Omron Sysmac Studio project AA_Festo (Sysmac Studio 1.60.0.64010, StandardProject)

# Controller Right_PLC: NX1P2-9B24DT1 version 1.42
Task PrimaryTask (priority 4, period or condition 4000): Main, Comunication_FINS
Library OEN_Communication_V1_0_22 1.0.22 (contents left out)
Library FINS_NX 1.1.0 (contents left out)

VAR_GLOBAL
    trama : ARRAY[0..3] OF OEN\Modbus\sModbusReq := [(Enable := True, NodeAdr := 1, FunctionCode := Fn15_WriteMultipleCoils, Read := (StartAddressRemote := 0, StartAddressLocal := 0, Count := 0), Write := (StartAddressRemote := 0, StartAddressLocal := 0, Count := 40)), (Enable := True, NodeAdr := 1, FunctionCode := Fn02_ReadDiscreteInputs, Read := (StartAddressRemote := 0, StartAddressLocal := 0, Count := 40), Write := (StartAddressRemote := 0, StartAddressLocal := 0, Count := 0)), (Enable := True, NodeAdr := 1, FunctionCode := Fn04_ReadInputRegisters, Read := (StartAddressRemote := 0, StartAddressLocal := 0, Count := 5), Write := (StartAddressRemote := 0, StartAddressLocal := 0, Count := 0)), (Enable := True, NodeAdr := 1, FunctionCode := Fn16_WriteMultipleRegisters, Read := (StartAddressRemote := 0, StartAddressLocal := 0, Count := 0), Write := (StartAddressRemote := 0, StartAddressLocal := 0, Count := 5))];
    out_Dig : ARRAY[0..99] OF BOOL;  (* Out_Digitais; [0] Emitter base; [1] Pneumatico inicio; [3] Motor Tapete; [4] Positioner Clamp; [5] Positioner raise (Stop Peça); [19] start button light A1; [8] Positioner Clamp extra; [9] Avanço Pneumatico Vácuo; [10] Baixa Pneumatico Vácuo; [11] Vácuo; [21] reset button light A1; [14] garra prende; [7] Emitter top; [15] Plataforma Frente; [16] Plataforma Tras; [20] stop button light A1; [17] Remover; [23] Start Button Light A2; [24] Stop Button Light A2; [25] Reset Button Light A2; [33] Reset Factory *)
    in_Dig : ARRAY[0..99] OF BOOL;  (* Entradas_Digitais; [1] Sensor Pneumático Trás; [0] Sensor Deteta Peça Base; [2] Sensor Pneumático Frente; [4] Sensor Inicio Tapete; [5] Sensor Leitura Cor; [8] Sensor Fim Tapete; [13] Sensor Vácuo Pneumatico cima; [10] Sensor Positioner clamp extra; [11] Sensor Vácuo Pneumatico  Frente; [6] Sensor Positioner raise; [23] Sensor Plataforma Trás; [17] Sensor Posição Recolha; [19] Sensor Posição Despeço Esquerda; [21] Sensor Garra Prende; [20] Sensor Posição Despejo Direita; [22] Sensor Plataforma Frente; [26] Stop Button A1; [25] Start Button A1; [14] Sensor Vácuo; [7] Sensor Positioner clamp; [12] Sensor Vácuo Pneumatico Trás; [18] Sensor Barra Início; [27] Reset Button A1; [29] Start Button A2; [30] Stop Button A2; [31] Reset Button A2; [33] Sensor Garra Cima; [34] Sensor Garra Baixo *)
    in_Analog : ARRAY[0..20] OF WORD;  (* Entradas_Analogicas *)
    out_analog : ARRAY[0..20] OF WORD;  (* Saidas_analogicas; [1] Garra y; [0] Garra x; [2] Garra Z *)
    A2_Start : BOOL;  (* at BuiltInIO://cpu/#0/Input_Bit_08 *)
    A2_Stop : BOOL;  (* at BuiltInIO://cpu/#0/Input_Bit_09 *)
    A2_Reset : BOOL;  (* at BuiltInIO://cpu/#0/Input_Bit_11 *)
    A2_Chave : BOOL;  (* at BuiltInIO://cpu/#0/Input_Bit_10 *)
    A2_S_PR : BOOL;  (* Sensor Posição Recolha; at BuiltInIO://cpu/#0/Input_Bit_00 *)
    A2_S_GC : BOOL;  (* Sensor Garra Cima; at BuiltInIO://cpu/#0/Input_Bit_05 *)
    A2_S_GP : BOOL;  (* Sensor Garra Prende; at BuiltInIO://cpu/#0/Input_Bit_06 *)
    A2_S_BI : BOOL;  (* Sensor Barra Início; at BuiltInIO://cpu/#0/Input_Bit_01 *)
    A2_S_GB : BOOL;  (* Sensor Garra Baixo; at BuiltInIO://cpu/#0/Input_Bit_04 *)
    A2_GP : BOOL;  (* Garra Prender; at BuiltInIO://cpu/#0/Output_Bit_02 *)
    A2_GE : BOOL;  (* Garra Esquerda; at BuiltInIO://cpu/#0/Output_Bit_00 *)
    A2_GB : BOOL;  (* Garra Baixo; at BuiltInIO://cpu/#0/Output_Bit_01 *)
    A2_S_PDD : BOOL;  (* Sensor Posição Despejo Direita; at BuiltInIO://cpu/#0/Input_Bit_02 *)
    A2_GD : BOOL;  (* Garra Direita; at BuiltInIO://cpu/#0/Output_Bit_03 *)
    A2_S_PDE : BOOL;  (* Sensor Posição Despeço Esquerda; at BuiltInIO://cpu/#0/Input_Bit_03 *)
    A2_PlT : BOOL;  (* Plataforma Tras; at BuiltInIO://cpu/#0/Output_Bit_09 *)
    A2_PlF : BOOL;  (* Plataforma Frente; at BuiltInIO://cpu/#0/Output_Bit_08 *)
    A2_S_PlF : BOOL;  (* Sensor Plataforma Frente; at BuiltInIO://cpu/#0/Input_Bit_12 *)
    A2_S_PlT : BOOL;  (* Sensor Plataforma Trás; at BuiltInIO://cpu/#0/Input_Bit_13 *)
    Emergency_right : BOOL;
    Emergency_claw_right : BOOL;
    Emergency_claw_left : BOOL;
    Emergency_paletization_back : BOOL;
    Emergency_paletization_front : BOOL;
    Emergency_claw_down : BOOL;
END_VAR
VAR_GLOBAL RETAIN
    Execute AT %D1.00 : BOOL := False;
END_VAR
VAR_GLOBAL
    Registers : ARRAY[0..499] OF WORD;
    NewValues : ARRAY[0..499] OF WORD := [16#CAFE, 16#DEAD, 498(16#0)];
END_VAR
VAR_GLOBAL RETAIN
    A1_MT AT %D1.02 : BOOL := False;
    cor_desejada_1 AT %D300.00 : BOOL := False;  (* published *)
    cor_desejada_2 AT %D300.01 : BOOL := False;  (* published *)
    cor_desejada_3 AT %D300.02 : BOOL := False;  (* published *)
    cor_desejada_4 AT %D300.03 : BOOL := False;  (* published *)
    cor_desejada AT %D300 : ARRAY[0..3] OF BOOL;
    espaco_posicao AT %D301 : ARRAY[0..3] OF BOOL;
    espaco_posicao_1 AT %D301.00 : BOOL := False;  (* published *)
    espaco_posicao_2 AT %D301.01 : BOOL := False;  (* published *)
    espaco_posicao_3 AT %D301.02 : BOOL := False;  (* published *)
    espaco_posicao_4 AT %D301.03 : BOOL := False;  (* published *)
    Cilindro_Base AT %D1.03 : BOOL;  (* published *)
    Cilindro_Tampa_Front AT %D1.04 : BOOL;  (* published *)
    Cilindro_Tampa_Back AT %D1.05 : BOOL;  (* published *)
    Cilindro_Tampa_Down AT %D1.06 : BOOL;  (* published *)
    Vácuo AT %D1.07 : BOOL;  (* published *)
    Travão_Montagem AT %D1.08 : BOOL;  (* published *)
    Tapete AT %D1.09 : BOOL;  (* published *)
END_VAR
VAR_GLOBAL
    Start : BOOL := False;  (* published *)
    Stop : BOOL := False;  (* published *)
    Reset : BOOL := False;  (* published *)
    Pick_and_Place_Right : BOOL := False;  (* published *)
    Pick_and_Place_Left : BOOL := False;  (* published *)
    Pick_and_Place_Down : BOOL := False;  (* published *)
    Garra_Pick_and_Place : BOOL := False;  (* published *)
    Paletização_Back : BOOL := False;  (* published *)
    Paletização_Front : BOOL := False;  (* published *)
END_VAR
VAR_GLOBAL RETAIN
    cor_automato_1 AT %D101 : ARRAY[0..3] OF BOOL;
END_VAR

PROGRAM Main
VAR
    ModBus_Client_PLC : OEN\Modbus\ModbusTCP_Client;
    E1 : ARRAY[0..20] OF BOOL;
    E0 : ARRAY[0..10] OF BOOL;
    timer_prende : TON;
    posicao_escolhida : INT;
    coloca_peca : BOOL;
    i : INT;
    init_program : BOOL;
    timer_emergency_down : TON;
    timer_emergency_left : TON;
    timer_emergency_right : TON;
    timer_emergency_paletization_back : TON;
    timer_emergency_paletization_front : TON;
END_VAR
VAR RETAIN
    D1_Word AT %D1 : WORD;
    A2_S_PR_A1 AT %D1.01 : BOOL;
    D100_Word AT %D100 : WORD;
    D101_Word AT %D101 : WORD;
END_VAR
VAR
    j : INT;
    timer_inicio_program : TON;
END_VAR
VAR RETAIN
    A1_S_IT AT %D100.04 : BOOL := False;  (* Sensor Inicio Tapete *)
    A1_S_C AT %D100.05 : BOOL := False;  (* Sensor Leitura Cor *)
    A1_S_FT AT %D100.06 : BOOL := False;  (* Sensor Fim Tapete *)
    A1_Start AT %D100.00 : BOOL := False;
    A1_Stop AT %D100.01 : BOOL := False;
    A1_Reset AT %D100.02 : BOOL := False;
    A1_MT AT %D1.02 : BOOL := False;
END_VAR
VAR
    timer_deita_fora : TON;
    timer_delay : TON;
END_VAR
VAR_EXTERNAL
    trama : ARRAY[0..3] OF OEN\Modbus\sModbusReq;
    out_Dig : ARRAY[0..99] OF BOOL;
    in_Dig : ARRAY[0..99] OF BOOL;
    in_Analog : ARRAY[0..20] OF WORD;
    out_analog : ARRAY[0..20] OF WORD;
    A2_S_PR : BOOL;
    A2_S_GP : BOOL;
    A2_S_BI : BOOL;
    A2_S_GC : BOOL;
    A2_GP : BOOL;
    A2_GE : BOOL;
    A2_GB : BOOL;
    A2_S_PDD : BOOL;
    A2_GD : BOOL;
    A2_Reset : BOOL;
    A2_S_PDE : BOOL;
    A2_PlT : BOOL;
    A2_PlF : BOOL;
    A2_S_PlF : BOOL;
    A2_S_PlT : BOOL;
    Emergency_claw_right : BOOL;
    Emergency_claw_left : BOOL;
    Emergency_paletization_back : BOOL;
    Emergency_paletization_front : BOOL;
    Emergency_claw_down : BOOL;
    A2_Start : BOOL;
    A2_Stop : BOOL;
    Execute : BOOL;
    NewValues : ARRAY[0..499] OF WORD;
    Registers : ARRAY[0..499] OF WORD;
    A2_S_GB : BOOL;
    cor_desejada : ARRAY[0..3] OF BOOL;
    espaco_posicao : ARRAY[0..3] OF BOOL;
    Start : BOOL;
    Stop : BOOL;
    Reset : BOOL;
    Pick_and_Place_Right : BOOL;
    Garra_Pick_and_Place : BOOL;
    Pick_and_Place_Left : BOOL;
    Pick_and_Place_Down : BOOL;
    Paletização_Front : BOOL;
    Paletização_Back : BOOL;
    A2_Chave : BOOL;
    cor_automato_1 : ARRAY[0..3] OF BOOL;
END_VAR
VAR
    _e1 : F_TRIG;
    _e2 : R_TRIG;
    _e3 : R_TRIG;
    _e4 : R_TRIG;
END_VAR

(* Section Comunication: ladder, written here as Structured Text *)

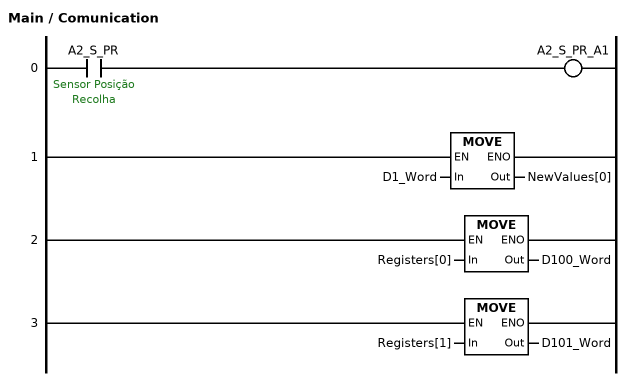
(* Rung 0 *)
A2_S_PR_A1 := A2_S_PR;
(* Rung 1 *)
NewValues[0] := D1_Word;
(* Rung 2 *)
D100_Word := Registers[0];
(* Rung 3 *)
D101_Word := Registers[1];

(* Section State_Machine: ladder, written here as Structured Text *)

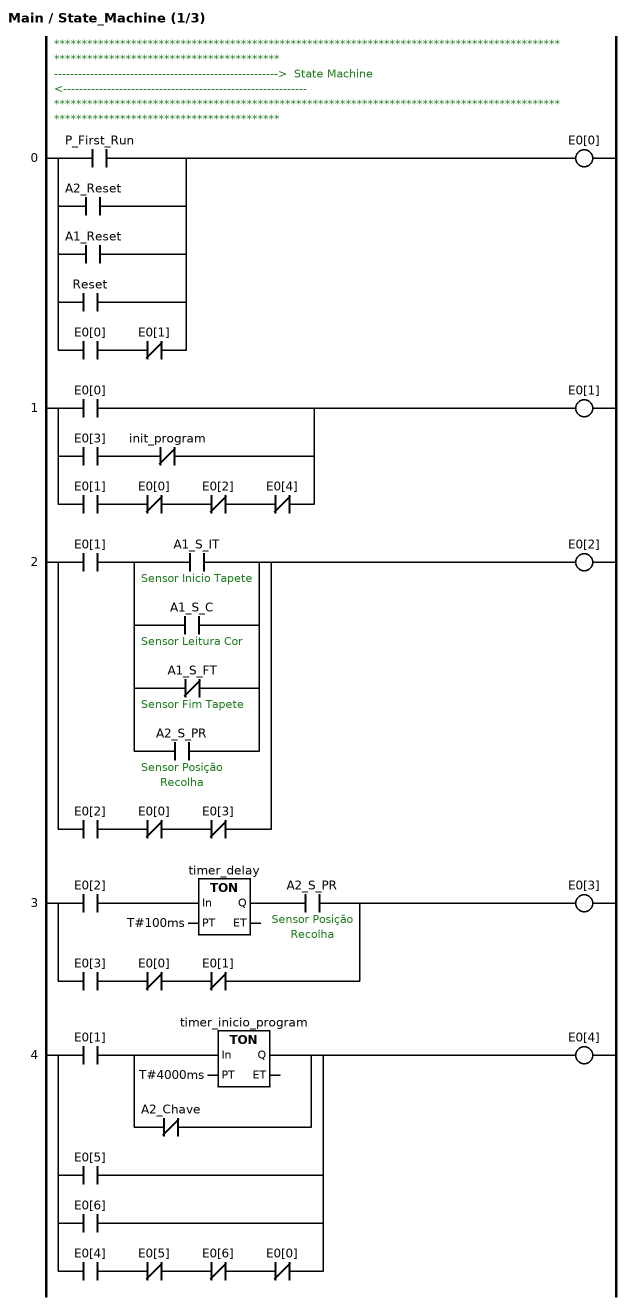
(* Rung 0: ************************************************************************************************************************************* / -------------------------------------------------------->  State Machine  <------------------------------------------------------------- / ************************************************************************************************************************************* *)
E0[0] := P_First_Run OR A2_Reset OR A1_Reset OR Reset OR (E0[0] AND NOT E0[1]);
(* Rung 1 *)
E0[1] := E0[0] OR (E0[3] AND NOT init_program) OR (E0[1] AND NOT E0[0] AND NOT E0[2] AND NOT E0[4]);
(* Rung 2 *)
E0[2] := (E0[1] AND (A1_S_IT OR A1_S_C OR NOT A1_S_FT OR A2_S_PR)) OR (E0[2] AND NOT E0[0] AND NOT E0[3]);
(* Rung 3 *)
timer_delay(In := E0[2], PT := T#100ms);
E0[3] := (timer_delay.Q AND A2_S_PR) OR (E0[3] AND NOT E0[0] AND NOT E0[1]);
(* Rung 4 *)
timer_inicio_program(In := E0[1], PT := T#4000ms);
E0[4] := timer_inicio_program.Q OR (E0[1] AND NOT A2_Chave) OR E0[5] OR E0[6] OR (E0[4] AND NOT E0[5] AND NOT E0[6] AND NOT E0[0]);

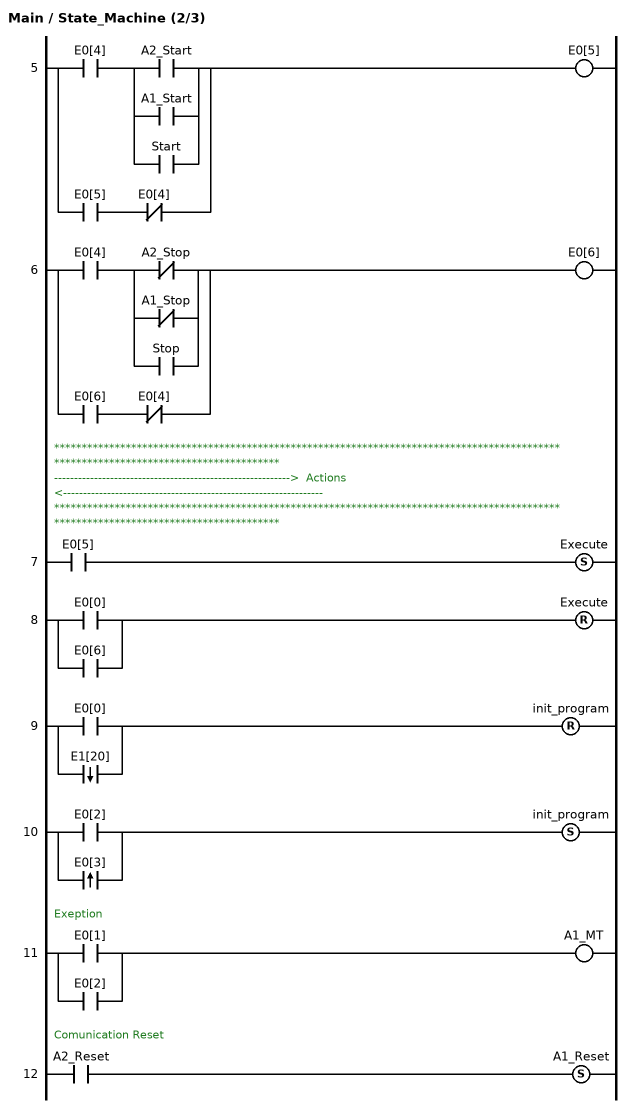
(* Rung 5 *)
E0[5] := (E0[4] AND (A2_Start OR A1_Start OR Start)) OR (E0[5] AND NOT E0[4]);
(* Rung 6 *)
E0[6] := (E0[4] AND (NOT A2_Stop OR NOT A1_Stop OR Stop)) OR (E0[6] AND NOT E0[4]);
(* Rung 7: ************************************************************************************************************************************* / ----------------------------------------------------------->  Actions  <----------------------------------------------------------------- / ************************************************************************************************************************************* *)
IF E0[5] THEN Execute := TRUE; END_IF;
(* Rung 8 *)
IF E0[0] OR E0[6] THEN Execute := FALSE; END_IF;
(* Rung 9 *)
_e1(CLK := E1[20]);
IF E0[0] OR _e1.Q THEN init_program := FALSE; END_IF;
(* Rung 10 *)
_e2(CLK := E0[3]);
IF E0[2] OR _e2.Q THEN init_program := TRUE; END_IF;
(* Rung 11: Exeption *)
A1_MT := E0[1] OR E0[2];
(* Rung 12: Comunication Reset *)
IF A2_Reset THEN A1_Reset := TRUE; END_IF;

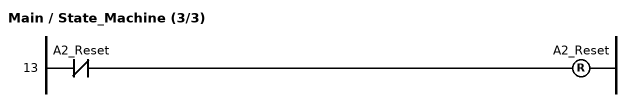
(* Rung 13 *)
IF NOT A2_Reset THEN A2_Reset := FALSE; END_IF;

(* Section Garra: ladder, written here as Structured Text *)

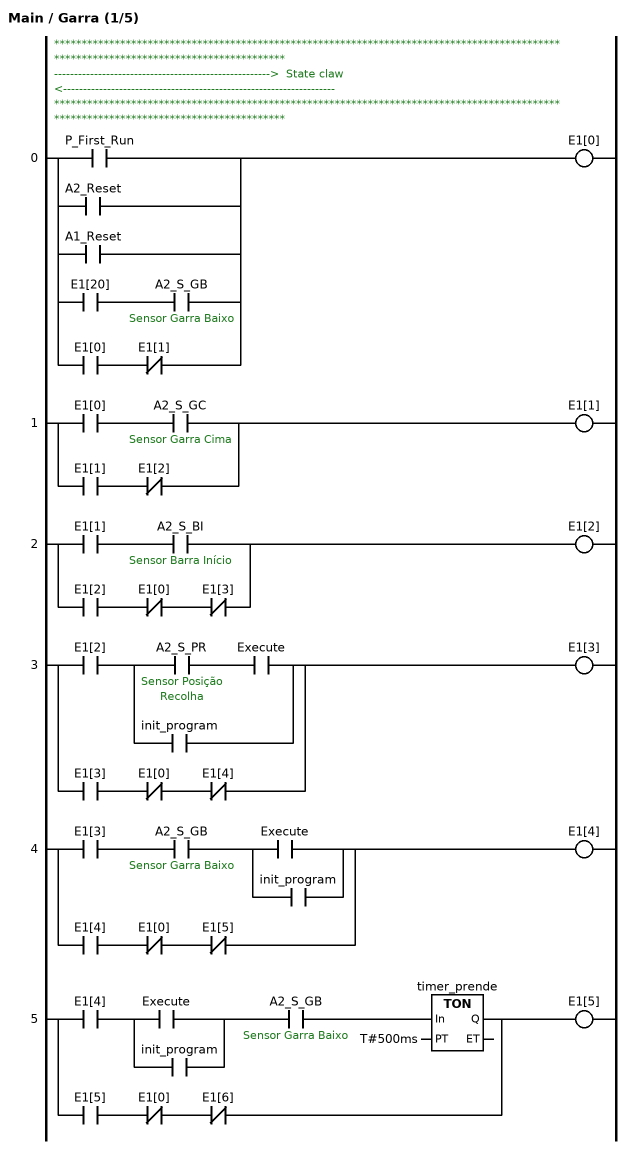
(* Rung 0: ************************************************************************************************************************************** / ------------------------------------------------------>  State claw  <-------------------------------------------------------------------- / ************************************************************************************************************************************** *)
E1[0] := P_First_Run OR A2_Reset OR A1_Reset OR (E1[20] AND A2_S_GB) OR (E1[0] AND NOT E1[1]);
(* Rung 1 *)
E1[1] := (E1[0] AND A2_S_GC) OR (E1[1] AND NOT E1[2]);
(* Rung 2 *)
E1[2] := (E1[1] AND A2_S_BI) OR (E1[2] AND NOT E1[0] AND NOT E1[3]);
(* Rung 3 *)
E1[3] := (E1[2] AND ((A2_S_PR AND Execute) OR init_program)) OR (E1[3] AND NOT E1[0] AND NOT E1[4]);
(* Rung 4 *)
E1[4] := (E1[3] AND A2_S_GB AND (Execute OR init_program)) OR (E1[4] AND NOT E1[0] AND NOT E1[5]);
(* Rung 5 *)
timer_prende(In := E1[4] AND (Execute OR init_program) AND A2_S_GB, PT := T#500ms);
E1[5] := timer_prende.Q OR (E1[5] AND NOT E1[0] AND NOT E1[6]);

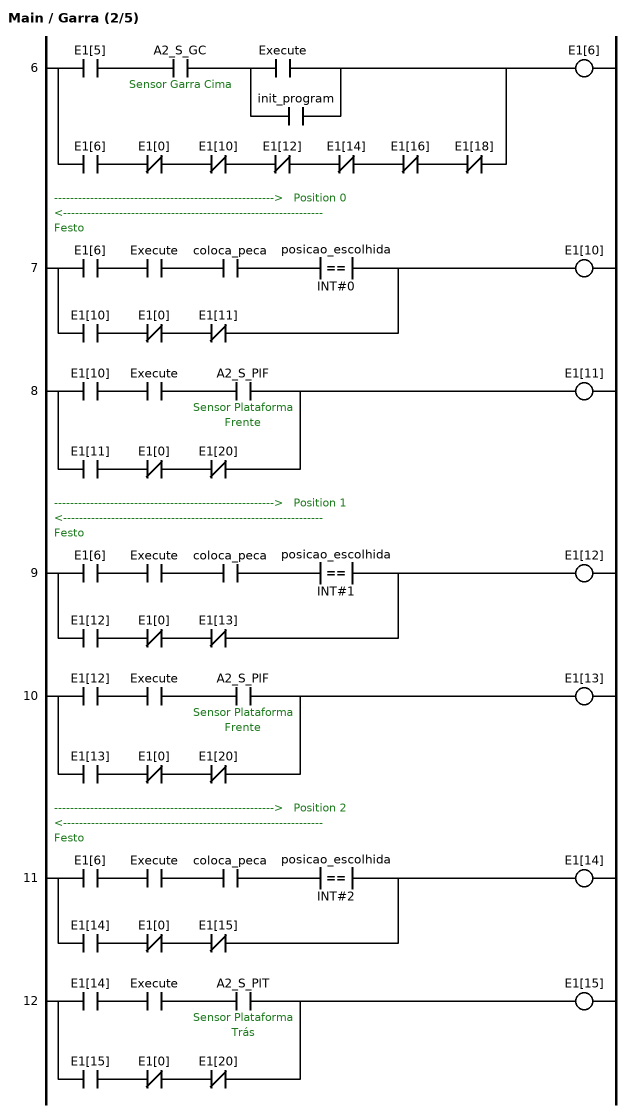
(* Rung 6 *)
E1[6] := (E1[5] AND A2_S_GC AND (Execute OR init_program)) OR (E1[6] AND NOT E1[0] AND NOT E1[10] AND NOT E1[12] AND NOT E1[14] AND NOT E1[16] AND NOT E1[18]);
(* Rung 7: ------------------------------------------------------->   Position 0   <----------------------------------------------------------------- / Festo *)
E1[10] := (E1[6] AND Execute AND coloca_peca AND (posicao_escolhida = INT#0)) OR (E1[10] AND NOT E1[0] AND NOT E1[11]);
(* Rung 8 *)
E1[11] := (E1[10] AND Execute AND A2_S_PlF) OR (E1[11] AND NOT E1[0] AND NOT E1[20]);
(* Rung 9: ------------------------------------------------------->   Position 1   <----------------------------------------------------------------- / Festo *)
E1[12] := (E1[6] AND Execute AND coloca_peca AND (posicao_escolhida = INT#1)) OR (E1[12] AND NOT E1[0] AND NOT E1[13]);
(* Rung 10 *)
E1[13] := (E1[12] AND Execute AND A2_S_PlF) OR (E1[13] AND NOT E1[0] AND NOT E1[20]);
(* Rung 11: ------------------------------------------------------->   Position 2   <----------------------------------------------------------------- / Festo *)
E1[14] := (E1[6] AND Execute AND coloca_peca AND (posicao_escolhida = INT#2)) OR (E1[14] AND NOT E1[0] AND NOT E1[15]);
(* Rung 12 *)
E1[15] := (E1[14] AND Execute AND A2_S_PlT) OR (E1[15] AND NOT E1[0] AND NOT E1[20]);

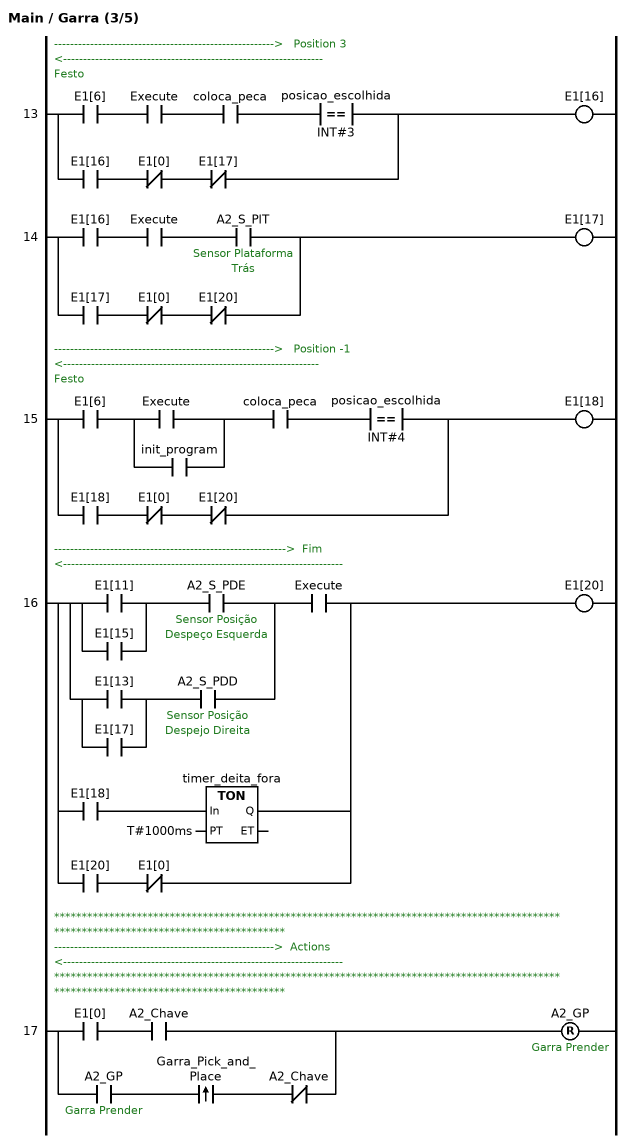
(* Rung 13: ------------------------------------------------------->   Position 3   <----------------------------------------------------------------- / Festo *)
E1[16] := (E1[6] AND Execute AND coloca_peca AND (posicao_escolhida = INT#3)) OR (E1[16] AND NOT E1[0] AND NOT E1[17]);
(* Rung 14 *)
E1[17] := (E1[16] AND Execute AND A2_S_PlT) OR (E1[17] AND NOT E1[0] AND NOT E1[20]);
(* Rung 15: ------------------------------------------------------->   Position -1   <---------------------------------------------------------------- / Festo *)
E1[18] := (E1[6] AND (Execute OR init_program) AND coloca_peca AND (posicao_escolhida = INT#4)) OR (E1[18] AND NOT E1[0] AND NOT E1[20]);
(* Rung 16: ---------------------------------------------------------->  Fim  <---------------------------------------------------------------------- *)
timer_deita_fora(In := E1[18], PT := T#1000ms);
E1[20] := ((((E1[11] OR E1[15]) AND A2_S_PDE) OR ((E1[13] OR E1[17]) AND A2_S_PDD)) AND Execute) OR timer_deita_fora.Q OR (E1[20] AND NOT E1[0]);
(* Rung 17: ************************************************************************************************************************************** / ------------------------------------------------------->  Actions <---------------------------------------------------------------------- / ************************************************************************************************************************************** *)
_e3(CLK := Garra_Pick_and_Place);
IF (E1[0] AND A2_Chave) OR (A2_GP AND _e3.Q AND NOT A2_Chave) THEN A2_GP := FALSE; END_IF;

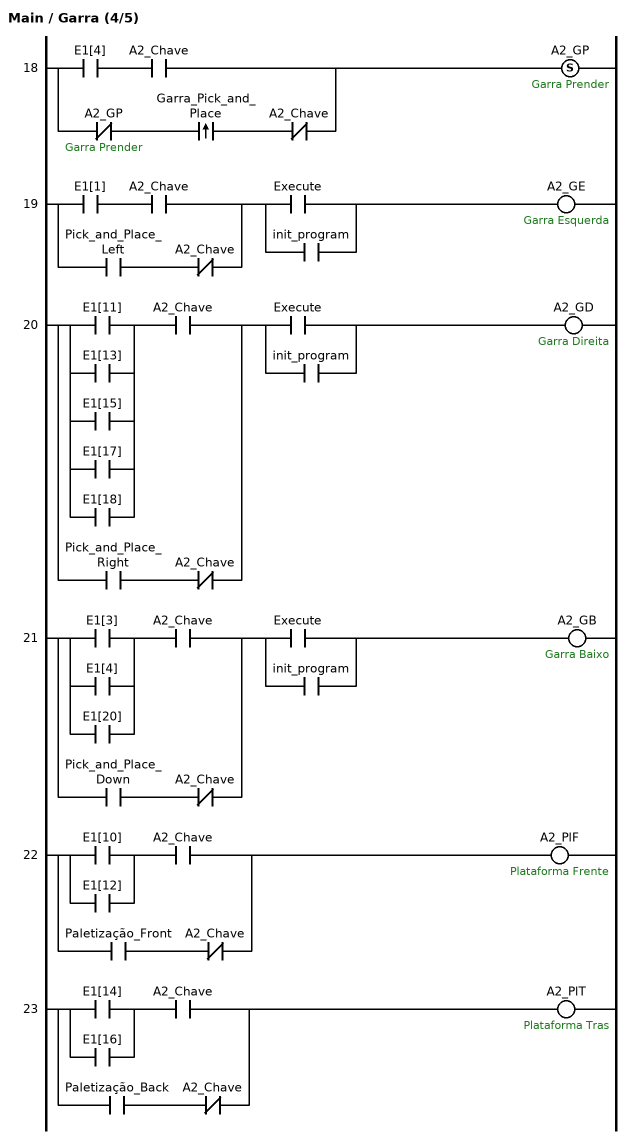
(* Rung 18 *)
_e4(CLK := Garra_Pick_and_Place);
IF (E1[4] AND A2_Chave) OR (NOT A2_GP AND _e4.Q AND NOT A2_Chave) THEN A2_GP := TRUE; END_IF;
(* Rung 19 *)
A2_GE := ((E1[1] AND A2_Chave) OR (Pick_and_Place_Left AND NOT A2_Chave)) AND (Execute OR init_program);
(* Rung 20 *)
A2_GD := (((E1[11] OR E1[13] OR E1[15] OR E1[17] OR E1[18]) AND A2_Chave) OR (Pick_and_Place_Right AND NOT A2_Chave)) AND (Execute OR init_program);
(* Rung 21 *)
A2_GB := (((E1[3] OR E1[4] OR E1[20]) AND A2_Chave) OR (Pick_and_Place_Down AND NOT A2_Chave)) AND (Execute OR init_program);
(* Rung 22 *)
A2_PlF := ((E1[10] OR E1[12]) AND A2_Chave) OR (Paletização_Front AND NOT A2_Chave);
(* Rung 23 *)
A2_PlT := ((E1[14] OR E1[16]) AND A2_Chave) OR (Paletização_Back AND NOT A2_Chave);

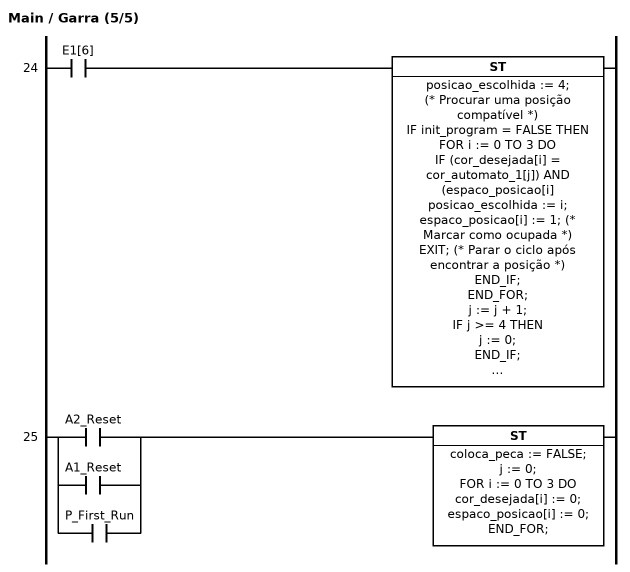
(* Rung 24 *)
IF E1[6] THEN
    posicao_escolhida := 4;
    
    (* Procurar uma posição compatível *)
    IF init_program = FALSE THEN
    	FOR i := 0 TO 3 DO
    	    IF (cor_desejada[i] = cor_automato_1[j]) AND (espaco_posicao[i] = 0) THEN
    			posicao_escolhida := i;
    	        espaco_posicao[i] := 1; (* Marcar como ocupada *)
    	        EXIT; (* Parar o ciclo após encontrar a posição *)
    	    END_IF;
    	END_FOR;
    	
    	j := j + 1;
    	IF j >= 4 THEN
    		j := 0;
    	END_IF;
    	
    END_IF;
    
    coloca_peca := TRUE;
END_IF;
(* Rung 25 *)
IF A2_Reset OR A1_Reset OR P_First_Run THEN
    coloca_peca := FALSE;
    j := 0;
    FOR i := 0 TO 3 DO
        cor_desejada[i] := 0;
        espaco_posicao[i] := 0;
    END_FOR;
END_IF;

(* Section Security: ladder, written here as Structured Text *)

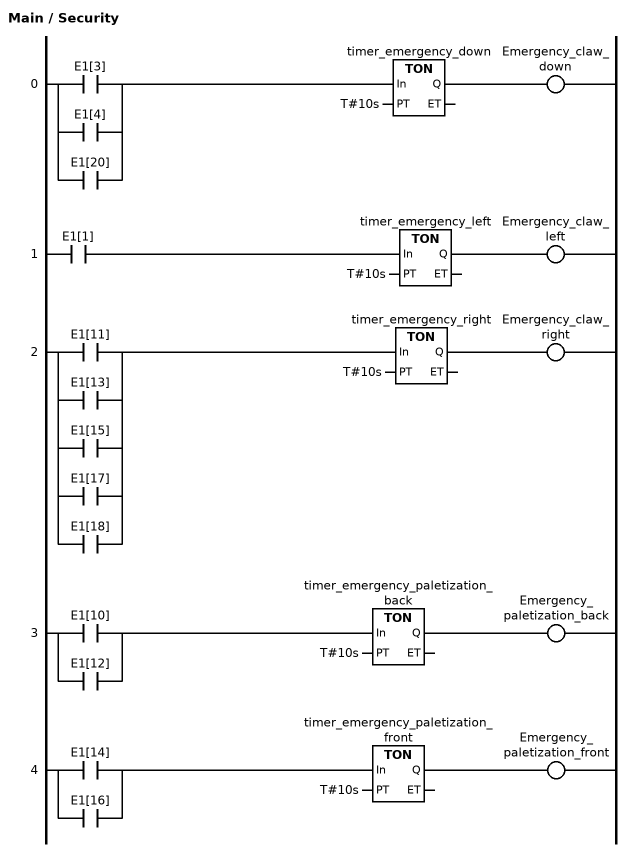
(* Rung 0 *)
timer_emergency_down(In := E1[3] OR E1[4] OR E1[20], PT := T#10s);
Emergency_claw_down := timer_emergency_down.Q;
(* Rung 1 *)
timer_emergency_left(In := E1[1], PT := T#10s);
Emergency_claw_left := timer_emergency_left.Q;
(* Rung 2 *)
timer_emergency_right(In := E1[11] OR E1[13] OR E1[15] OR E1[17] OR E1[18], PT := T#10s);
Emergency_claw_right := timer_emergency_right.Q;
(* Rung 3 *)
timer_emergency_paletization_back(In := E1[10] OR E1[12], PT := T#10s);
Emergency_paletization_back := timer_emergency_paletization_back.Q;
(* Rung 4 *)
timer_emergency_paletization_front(In := E1[14] OR E1[16], PT := T#10s);
Emergency_paletization_front := timer_emergency_paletization_front.Q;
END_PROGRAM

PROGRAM Comunication_FINS
VAR
    Write : BOOL;
    FINS_Write_Inst : FINS_Write;
    DestNetAddr : FINS\sNetAddr;
    DestArea : FINS\eArea;
    DestAddr : UINT;
    WriteDone : BOOL;
    Error : BOOL;
    ErrorID : WORD;
    SelectPLC : BOOL;
    rep : ARRAY[0..2000] OF BYTE;
    FINScode : WORD;
    Read : BOOL;
    FINS_Read_Inst : FINS_Read;
    SrcNetAddr : FINS\sNetAddr;
    ReadDone : BOOL;
    Read_Error : BOOL;
    Read_ErrorID : WORD;
    Read_FINScode : WORD;
    RcvSize : UINT;
    Diffup : R_TRIG;
    DiffDown : F_TRIG;
    TesteCom : WORD;
END_VAR
VAR_EXTERNAL
    Registers : ARRAY[0..499] OF WORD;
    NewValues : ARRAY[0..499] OF WORD;
END_VAR

(* Section FINS_Comms: ladder, written here as Structured Text *)

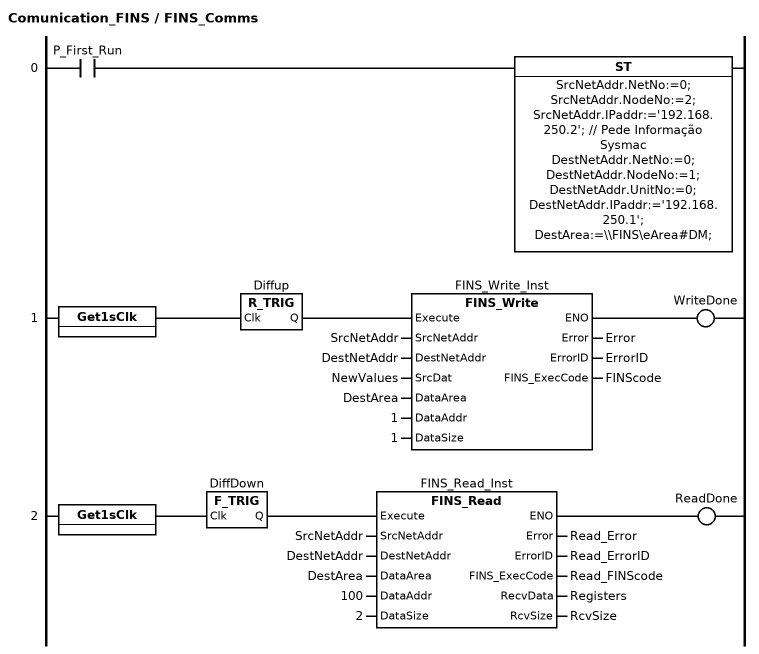
(* Rung 0 *)
IF P_First_Run THEN
    SrcNetAddr.NetNo:=0;
    SrcNetAddr.NodeNo:=2;
    SrcNetAddr.IPaddr:='192.168.250.2'; // Pede Informação Sysmac
    DestNetAddr.NetNo:=0;
    DestNetAddr.NodeNo:=1;
    DestNetAddr.UnitNo:=0;
    DestNetAddr.IPaddr:='192.168.250.1';
    DestArea:=\\FINS\eArea#DM;
END_IF;
(* Rung 1 *)
Diffup(Clk := Get1sClk());
FINS_Write_Inst(Execute := Diffup.Q, SrcNetAddr := SrcNetAddr, DestNetAddr := DestNetAddr, SrcDat := NewValues, DataArea := DestArea, DataAddr := 1, DataSize := 1, Error => Error, ErrorID => ErrorID, FINS_ExecCode => FINScode);
WriteDone := FINS_Write_Inst.ENO;
(* Rung 2 *)
DiffDown(Clk := Get1sClk());
FINS_Read_Inst(Execute := DiffDown.Q, SrcNetAddr := SrcNetAddr, DestNetAddr := DestNetAddr, DataArea := DestArea, DataAddr := 100, DataSize := 2, Error => Read_Error, ErrorID => Read_ErrorID, FINS_ExecCode => Read_FINScode, RecvData => Registers, RcvSize => RcvSize);
ReadDone := FINS_Read_Inst.ENO;
END_PROGRAM

# Device HMI_NA5_0 (NA): not converted